# B&R Automation Studio project AsProject
Automation Studio 6.5.1.7; Starter Automation Studio project.; technology packages: OpcUaCs 6.6.1

## Configuration ARM

CPU X20CP0484, AutomationRuntime 6.6.2, Build 11.3.0, Vc 6.0.0

### Task classes (Cpu.sw)
```
Libraries: ArEventLog, AsARCfg, AsArProf, AsBrMath, AsBrStr, AsBrWStr, AsEPL, AsGuard, AsHttp, AsIO, AsIOAcc, AsIODiag, AsIOTime, AsMem, AsSem, AsTCP, AsUDP, AsUSB, AsXml, AsZip, astime, brsystem, DataObj, dvframe, FileIO, LoopConR, MTBasics, MTLookUp, MTTypes, operator, runtime, standard, sys_lib, Persist
```

### Hardware
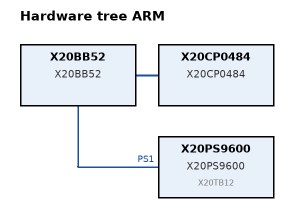
```
X20BB52 : X20BB52 v1.2.0.0
X20CP0484 : X20CP0484 v1.8.1.0  [SL -> X20BB52.SL1]
  Connector IF2:
    ActivateDevice = 1
  ConfigurationID = AsProject_ARM
  PermanentPvSize = 50000
  RemanentGlobalPvSize = 10000
  TimerDeviceType = SWIOTIMER
  Cyclic1Duration = 10000
  Cyclic1Tolerance = 10000
  Cyclic2Duration = 20000
  Cyclic2Tolerance = 20000
  Cyclic3Duration = 50000
  Cyclic3Tolerance = 50000
  Cyclic4Duration = 100000
  Cyclic4Tolerance = 100000
  Cyclic5Duration = 200000
  Cyclic5Tolerance = 200000
  Cyclic6Duration = 500000
  Cyclic6Tolerance = 500000
  Cyclic7Duration = 1000000
  Cyclic7Tolerance = 1000000
  Cyclic8Duration = 10000
  Cyclic8Tolerance = 30000000
  FileDevice1
  FileDeviceName1 = USER
  FileDevicePath1 = USER_PATH
X20PS9600 : X20PS9600 v1.6.2.0  [PS -> X20BB52.PS1; SS1 -> X20TB12.SS]
X20TB12 : X20TB12 v1.0.0.0
```

### BRRole.brrole - X20CP0484/AccessAndSecurity/UserRoleSystem/BRRole.brrole
```
Element BR_Anonymous (Type=BRRole)
Element BR_Engineer (Type=BRRole)
Element BR_Observer (Type=BRRole)
Element BR_SafetyAdmin (Type=BRRole)
Element BR_SecurityAdmin (Type=BRRole)
```

- Physical/ARM/X20CP0484/IoMap.iom: same as Physical/ARM/X20CP0484/Cpu.per
- Physical/ARM/X20CP0484/PvMap.vvm: same as Physical/ARM/X20CP0484/Cpu.per
- Safety project (password-protected, skipped)

## Configuration Intel

CPU 5APC4100.TGL1-000, AutomationRuntime 6.6.2, Build 11.3.0, Vc 6.0.0

### Task classes (Cpu.sw)
```
Binaries: udbdef, TCData, FWRules, ashwd, ashwac, User, sysconf, asfw, arconfig, iomap, Role
Libraries: ArEventLog, AsARCfg, AsArProf, AsBrMath, AsBrStr, AsEPL, AsGuard, AsHttp, AsIO, AsIOAcc, AsIODiag, AsIOTime, AsMem, AsSem, AsTCP, astime, AsUDP, AsUSB, AsXml, AsZip, brsystem, DataObj, dvframe, FileIO, operator, runtime, standard, sys_lib, AsBrWStr, MTTypes, MTBasics, LoopConR, MTLookUp, Persist
```

### Hardware
```
5AC901.IPLK-00 : 5AC901.IPLK-00 v2.1.0.0  [SS -> 5APC4100_TGL1_000.SS2]
  Connector IF1:
    DNAConfiguration = manual
5APC4100_TGL1_000 : 5APC4100.TGL1-000 v1.3.1.0
  Connector IF3:
    AssignedOperatingSystem = ARemb
    ActivateDevice = 1
  Connector IF4:
    AssignedOperatingSystem = ARemb
    ActivateDevice = 1
  Connector IF5:
    AssignedOperatingSystem = ARemb
    ActivateDevice = 1
  Connector IF6:
    AssignedOperatingSystem = ARemb
    ActivateDevice = 1
  Connector IF7:
    AssignedOperatingSystem = ARemb
  Connector IF8:
    AssignedOperatingSystem = ARemb
  Connector IF9:
    AssignedOperatingSystem = ARemb
  Connector IF10:
    AssignedOperatingSystem = ARemb
  Connector IF11:
    AssignedOperatingSystem = ARemb
  Connector IF12:
    AssignedOperatingSystem = ARemb
  ConfigurationID = AsProject_Intel
  UserPartitionSize = 300
  Simulation = 1
  UserRamDevice = PCI.2.IPLK.SRAM
  UserRamSize = 500000
  RemMemDevice = PCI.2.IPLK.SRAM
  RemMemSize = 120000
  PermanentPvSize = 10000
  RemanentGlobalPvSize = 105000
  VolatileGlobalPvSize = 1000000
  TimerDeviceType = EPLX2X
  TimerDevice = 5AC901.IPLK-00.IF1
  IdleTaskClass = 3
  TaskClassIdleTime = 8000
  Cyclic1Duration = 2000
  Cyclic1Tolerance = 0
  Cyclic2Duration = 10000
  Cyclic3Duration = 20000
  Cyclic3Tolerance = 40000
  FileDevice1
  FileDeviceName1 = USER
  FileDevicePath1 = USER_PATH
  TimeZone = 25
  ActivateFtpServer = 1
  FtpUser1
  FtpUsername1 = dev
  FtpUserPassword1 = o33x/UifGm0mfwtuaZAada64hc3m8aosihbfwQCh3ow=  // dev
  FtpUserSalt1 = 2jAdfp5W
  FTPAccessRight1 = 0
  FTPdevice1 = ALL
  ActivateWebServer = 1
  ActivateSdm = 1
  SdmColor = colorRGB
```

- Physical/Intel/5APC4100_TGL1_000/AccessAndSecurity/UserRoleSystem/BRRole.brrole: same as Physical/ARM/X20CP0484/AccessAndSecurity/UserRoleSystem/BRRole.brrole
- Physical/Intel/5APC4100_TGL1_000/IoMap.iom: same as Physical/Intel/5APC4100_TGL1_000/Cpu.per
- Physical/Intel/5APC4100_TGL1_000/PvMap.vvm: same as Physical/Intel/5APC4100_TGL1_000/Cpu.per
## Logical view

Binary libraries used (declarations not repeated): ArEventLog, AsARCfg, AsArProf, AsBrMath, AsBrStr, AsEPL, AsGuard, AsHttp, AsIO, AsIOAcc, AsIODiag, AsIOTime, AsMem, AsSem, astime, AsTCP, AsUDP, AsUSB, AsXml, AsZip, brsystem, DataObj, dvframe, FileIO, operator, runtime, standard, sys_lib, AsBrWStr, MTTypes 6.0.0, MTBasics 6.4.0, LoopConR 6.0.0, MTLookUp 6.4.0, Persist
